{attribute 'GeneratedUsingTerminal: EL3202-0030-0022'}
{attribute addProperty BoxType "EL3202-0030-0022"}
{attribute addProperty Id "StatusAT %I*Status_F2CE6D917ValueAT %I*INT2"}
{attribute addProperty CRC "1245267073"}
{attribute addProperty Size "9"}
TYPE RTD_Inputs_Channel_4A394481 :
STRUCT
	{attribute addProperty Name "Status"}
	Status AT %I* : Status_F2CE6D91;
	{attribute addProperty Name "Value"}
	Value AT %I* : INT;
END_STRUCT
END_TYPE

(* stored: Version 1.2.0.0, ProductVersion 3.1.4024.9
   DUT RTD_Inputs_Channel_4A394481: Id {8134e550-a7a0-4ef2-adb9-3a37802f5bc2} *)
